KUKA KRL program: command_handler.src, command_handler.dat

--- command_handler.src ---
&ACCESS RVP
&PARAM EDITMASK = *
&PARAM TEMPLATE = C:\KRC\Roboter\Template\vorgabe
DEF command_handler()

   ; Software License Agreement (BSD License)
   ;
   ; Copyright (c) 2022, Kuka Robotics Corp
   ; All rights reserved.
   ;
   ; Redistribution and use in source and binary forms, with or without
   ; modification, are permitted provided that the following conditions are met:
   ;
   ;      * Redistributions of source code must retain the above copyright
   ;        notice, this list of conditions and the following disclaimer.
   ;      * Redistributions in binary form must reproduce the above copyright
   ;        notice, this list of conditions and the following disclaimer in the
   ;        documentation and/or other materials provided with the distribution.
   ;      * Neither the name of the copyright holder, nor the names of its
   ;        contributors may be used to endorse or promote products derived
   ;        from this software without specific prior written permission.
   ;
   ; THIS SOFTWARE IS PROVIDED BY THE COPYRIGHT HOLDERS AND CONTRIBUTORS "AS IS"
   ; AND ANY EXPRESS OR IMPLIED WARRANTIES, INCLUDING, BUT NOT LIMITED TO, THE
   ; IMPLIED WARRANTIES OF MERCHANTABILITY AND FITNESS FOR A PARTICULAR PURPOSE
   ; ARE DISCLAIMED. IN NO EVENT SHALL THE COPYRIGHT OWNER OR CONTRIBUTORS BE
   ; LIABLE FOR ANY DIRECT, INDIRECT, INCIDENTAL, SPECIAL, EXEMPLARY, OR
   ; CONSEQUENTIAL DAMAGES (INCLUDING, BUT NOT LIMITED TO, PROCUREMENT OF
   ; SUBSTITUTE GOODS OR SERVICES; LOSS OF USE, DATA, OR PROFITS; OR BUSINESS
   ; INTERRUPTION) HOWEVER CAUSED AND ON ANY THEORY OF LIABILITY, WHETHER IN
   ; CONTRACT, STRICT LIABILITY, OR TORT (INCLUDING NEGLIGENCE OR OTHERWISE)
   ; ARISING IN ANY WAY OUT OF THE USE OF THIS SOFTWARE, EVEN IF ADVISED OF THE
   ; POSSIBILITY OF SUCH DAMAGE.

END

GLOBAL DEF HandleCommand(cmd:IN)
   DECL Command cmd
   DECL CMDType cmd_enum
   DECL BOOL cmd_success
   DECL ControlMode mode

   cmd_enum = ParseCommand(cmd.cmd_str[])

   IF cmd_enum == #CMD_NONE THEN
      ; If nothing was received, just RETURN
      RETURN
   ENDIF

   IF ValidateCommand(cmd_enum) THEN

      SWITCH cmd_enum
         CASE #CMD_INVALID
            SetEvent(#Invalid)
         CASE #CMD_CON
            SetEvent(#Connected)
         CASE #CMD_START
            cmd_success = StartProgram(GetProgName(GetControlMode()))
            IF cmd_success THEN
               driver_state = #Active
               SetEvent(#Started)
            ELSE
               SetEvent(#Error)
            ENDIF
         CASE #CMD_CANCEL
            cmd_success = CancelProgram()
            IF cmd_success THEN
               driver_state = #Initialized
               SetControlMode(#Inactive)
               SetEvent(#Cancelled)
            ELSE
               SetEvent(#Error)
            ENDIF
         CASE #CMD_RESET
            cmd_success = ResetProgram()
            IF cmd_success THEN
               driver_state = #Inactive
               SetEvent(#ResetOK)
            ELSE
               SetEvent(#Error)
            ENDIF
         CASE #CMD_CHANGE
            SWITCH cmd.control_mode
               CASE 1
                  mode = #JointPosition
               CASE 5
                  mode = #CartPosition
               DEFAULT
                  SetEvent(#Error)
                  RETURN
            ENDSWITCH
            SetControlMode(mode) ; TODO
            driver_state = #Inactive
            SetEvent(#SwitchOK)
      ENDSWITCH
   ELSE
      SetEvent(#Invalid)
      MsgNotify("Invalid transition requested")
   ENDIF

END

DEFFCT CMDType ParseCommand(cmd[]:IN)
   CHAR cmd[]

   IF (StrComp(cmd[], "CON", #NOT_CASE_SENS)) THEN
      RETURN #CMD_CON
   ENDIF

   IF (StrComp(cmd[], "START", #NOT_CASE_SENS)) THEN
      RETURN #CMD_START
   ENDIF

   IF (StrComp(cmd[], "RESET", #NOT_CASE_SENS)) THEN
      RETURN #CMD_RESET
   ENDIF

   IF (StrComp(cmd[], "CANCEL", #NOT_CASE_SENS)) THEN
      RETURN #CMD_CANCEL
   ENDIF

   IF (StrComp(cmd[], "CHANGE", #NOT_CASE_SENS)) THEN
      RETURN #CMD_CHANGE
   ENDIF

   IF (StrComp(cmd[], "None", #NOT_CASE_SENS)) THEN
      RETURN #CMD_NONE
   ENDIF

   RETURN #CMD_INVALID
ENDFCT

DEFFCT BOOL ValidateCommand(cmd:IN)
   DECL CMDType cmd
   CHAR cmdString[16]
   CHAR stateString[16]

   ; Debug messages
   cmdString[] = CommandToString(cmd)
   stateString[] = DriverStateToString(driver_state)
   MsgNotifyTextPar("Got command %1 while in %2.", "CommandHandler", 0, cmdString[], stateString[])

   SWITCH driver_state
      CASE #Initialized
         RETURN (cmd == #CMD_CON) OR (cmd == #CMD_CHANGE)

      CASE #Inactive
         RETURN (cmd == #CMD_START) OR (cmd == #CMD_CHANGE) OR (cmd == #CMD_CANCEL)

      CASE #Active
         RETURN (cmd == #CMD_CANCEL) OR (cmd == #CMD_RESET)
   ENDSWITCH

   RETURN FALSE
ENDFCT

DEFFCT CHAR [16] CommandToString(command: IN)
   DECL CMDType command
   SWITCH command
      CASE #CMD_NONE
         RETURN "None"
      CASE #CMD_CON
         RETURN "Connect"
      CASE #CMD_START
         RETURN "Start"
      CASE #CMD_RESET
         RETURN "Reset"
      CASE #CMD_CANCEL
         RETURN "Cancel"
      CASE #CMD_CHANGE
         RETURN "Change"
      CASE #CMD_INVALID
         RETURN "Invalid"
   ENDSWITCH
ENDFCT

DEFFCT CHAR [16] DriverStateToString(driverState: IN)
   DECL DriverState driverState
   SWITCH driverState
      CASE #Initialized
         RETURN "Initialized"
      CASE #Inactive
         RETURN "Inactive"
      CASE #Active
         RETURN "Active"
   ENDSWITCH
ENDFCT

GLOBAL DEF SetDriverState(state: IN)
   DECL DriverState state
   driver_state = state
END

--- command_handler.dat ---
&ACCESS RV
&REL 11735
&PARAM DISKPATH = KRC:\R1\Program\ROS
DEFDAT command_handler PUBLIC
    ; FOLD Custom enumerations
    CONST INT STATE_COUNT = 3
    GLOBAL ENUM DriverState INITIALIZED, INACTIVE, ACTIVE

    GLOBAL ENUM EventType NONE, INVALID, STARTED, STOPPED, CANCELLED, RESET_OK, ERROR, CONNECTED, SWITCH_OK, DRIVES_TURNED_ON, DRIVES_TURNED_OFF

    CONST INT CMD_COUNT = 9
    GLOBAL ENUM CMDType CMD_NONE, CMD_CON, CMD_START, CMD_RESET, CMD_CANCEL, CMD_CHANGE, CMD_INVALID, CMD_DRIVES_ON, CMD_DRIVES_OFF, CMD_CHANGE_OP_MODE

    GLOBAL CONST INT CONTROL_MODE_COUNT = 2
    GLOBAL ENUM ControlMode INACTIVE, JOINT_POSITION, CART_POSITION
    ; ENDFOLD

    ; FOLD Custom structure types
    GLOBAL STRUC Command CHAR cmd_str[32], INT control_mode, CHAR operation_mode[32]
    STRUC StringCommandPair CHAR cmd_string[32], CMDType cmd_type
    STRUC StringStatePair CHAR state_string[32], DriverState state
    STRUC StateIntPair DriverState state, INT valid_count
    ; ENDFOLD

    DECL DriverState current_driver_state = #INITIALIZED

    ; FOLD Constants for mapping strings to command types
    DECL CONST StringCommandPair STRING_COMMAND_PAIRS[9]
    STRING_COMMAND_PAIRS[1] = { cmd_string[] "CON", cmd_type #CMD_CON }
    STRING_COMMAND_PAIRS[2] = { cmd_string[] "START", cmd_type #CMD_START }
    STRING_COMMAND_PAIRS[3] = { cmd_string[] "RESET", cmd_type #CMD_RESET }
    STRING_COMMAND_PAIRS[4] = { cmd_string[] "CANCEL", cmd_type #CMD_CANCEL }
    STRING_COMMAND_PAIRS[5] = { cmd_string[] "CHANGE", cmd_type #CMD_CHANGE }
    STRING_COMMAND_PAIRS[6] = { cmd_string[] "NONE", cmd_type #CMD_NONE }
    STRING_COMMAND_PAIRS[7] = { cmd_string[] "DRIVES_ON", cmd_type #CMD_DRIVES_ON }
    STRING_COMMAND_PAIRS[8] = { cmd_string[] "DRIVES_OFF", cmd_type #CMD_DRIVES_OFF }
    STRING_COMMAND_PAIRS[9] = { cmd_string[] "CHANGE_OP_MODE", cmd_type #CMD_CHANGE_OP_MODE }
    ; ENDFOLD

    ; FOLD Constants for mapping strings to driver states
    DECL CONST StringStatePair STRING_STATE_PAIRS[3]
    STRING_STATE_PAIRS[1] = { state_string "INITIALIZED", state #INITIALIZED }
    STRING_STATE_PAIRS[2] = { state_string "INACTIVE", state #INACTIVE }
    STRING_STATE_PAIRS[3] = { state_string "ACTIVE", state #ACTIVE }
    ; ENDFOLD

    ; FOLD Constants for mapping driver states to valid commands
    DECL CONST StateIntPair STATE_VALID_COUNTS[3]
    STATE_VALID_COUNTS[1] = { state #INITIALIZED, valid_count 4 }
    STATE_VALID_COUNTS[2] = { state #INACTIVE, valid_count 5 }
    STATE_VALID_COUNTS[3] = { state #ACTIVE, valid_count 2 }

    DECL CONST CMDType INIT_VALID_COMMANDS[16]
    INIT_VALID_COMMANDS[1] = #CMD_CON
    INIT_VALID_COMMANDS[2] = #CMD_CHANGE
    INIT_VALID_COMMANDS[3] = #CMD_DRIVES_ON
    INIT_VALID_COMMANDS[4] = #CMD_DRIVES_OFF

    DECL CONST CMDType INACTIVE_VALID_COMMANDS[16]
    INACTIVE_VALID_COMMANDS[1] = #CMD_START
    INACTIVE_VALID_COMMANDS[2] = #CMD_CHANGE
    INACTIVE_VALID_COMMANDS[3] = #CMD_CANCEL
    INACTIVE_VALID_COMMANDS[4] = #CMD_DRIVES_ON
    INACTIVE_VALID_COMMANDS[5] = #CMD_DRIVES_OFF

    DECL CONST CMDType ACTIVE_VALID_COMMANDS[16]
    ACTIVE_VALID_COMMANDS[1] = #CMD_CANCEL
    ACTIVE_VALID_COMMANDS[2] = #CMD_RESET
    ; ENDFOLD
ENDDAT
